TYPE ST_MV_EMAG_VLC100Y_Zustand :
STRUCT
	Kuehlung_Anford		: BOOL;
	Betrieb				: BOOL;

	Kommunikation		: BOOL;

	Stoerung			: BOOL;
	Stoerung_Code		: WORD;

	Warnung				: BOOL;
	Warnung_Code		: WORD;

	Status				: SINT;
END_STRUCT
END_TYPE

(* stored: Version 1.1.0.1, ProductVersion 3.1.4024.9
   DUT ST_MV_EMAG_VLC100Y_Zustand: Id {b0a1d3b1-13fc-46f7-8ba1-5ea7c848e173} *)
